// TIA Portal V17 export
// export: Created 2024-08-20T13:26:08.3005341Z, ExportSetting WithDefaults, DisplayName Totally Integrated Automation Portal, DisplayVersion V17 Update 4, DisplayName TIA Portal Openness, DisplayVersion V17 Update 4, DisplayName TIA Portal Version Control Interface, DisplayVersion V17, DisplayName STEP 7 Professional, DisplayVersion V17 Update 4, DisplayName STEP 7 Safety, DisplayVersion V17, DisplayName WinCC Advanced, DisplayVersion V17 Update 4
FUNCTION_BLOCK "INTPRO"   // FB202, LAD
{ S7_Optimized_Access := 'FALSE' }
VERSION : 0.1
// stored: AutoNumber true, IsIECCheckEnabled false, SetENOAutomatically false, UDAEnableTagReadback false
   VAR DB_SPECIFIC
      EE_P_NIV : Bool;   // HAILITA BOMBA PRINCIPAL PELO NÍVEL
      EE_C1_NIV : Bool;   // HAILITA BOMBA COMPLEMENTAR 1 PELO NÍVEL
      EE_C2_NIV : Bool;   // HAILITA BOMBA COMPLEMENTAR 2 PELO NÍVEL
      EE_P_LS : Bool;   // HAILITA BOMBA PRINCIPAL PELAS BÓIAS
      EE_C1_LS : Bool;   // HAILITA BOMBA COMLEMENTAR 1 PELAS BÓIAS
      EE_C2_LS : Bool;   // HAILITA BOMBA COMPLEMENTAR 2 PELAS BÓIAS
      HAB_P_EE : Bool;   // LIGA BOMBA PRINCIPAL DA ELEVATÓRIA
      HAB_C1_EE : Bool;   // LIGA BOMBA COMPLEMENTAR 1 DA ELEVATÓRIA
      HAB_C2_EE : Bool;   // LIGA BOMBA COMPLEMENTAR 2 DA ELEVATÓRIA
      AUXP01 : Bool;
      BS01OK : Bool;
      BS02OK : Bool;
      BS03OK : Bool;
      L_BS01 : Bool;
      L_BS02 : Bool;
      L_BS03 : Bool;
      AUXP02 : Bool;
      AUXP03 : Bool;
      AUXP04 : Bool;
      AUXP05 : Bool;
      AUXP06 : Bool;
      AUXP07 : Bool;
      ETBS01_T001 : Int;
      ETBS02_T001 : Int;
      ETBS03_T001 : Int;
      BS01TO : Int;
      BS02TO : Int;
      BS03TO : Int;
      BS01TEOK : DInt;
      BS02TEOK : DInt;
      BS03TEOK : DInt;
      TE00 { S7_SetPoint := 'True'} : IEC_TIMER;
   END_VAR
   VAR
      RODEE { S7_SetPoint := 'True'} : "ROD4";
   END_VAR
   VAR_TEMP
      T011S : Int;
      ET_TE00 : Time;
   END_VAR
BEGIN

REGION Network 1: Alarme falha de sinal transmissor de nivel
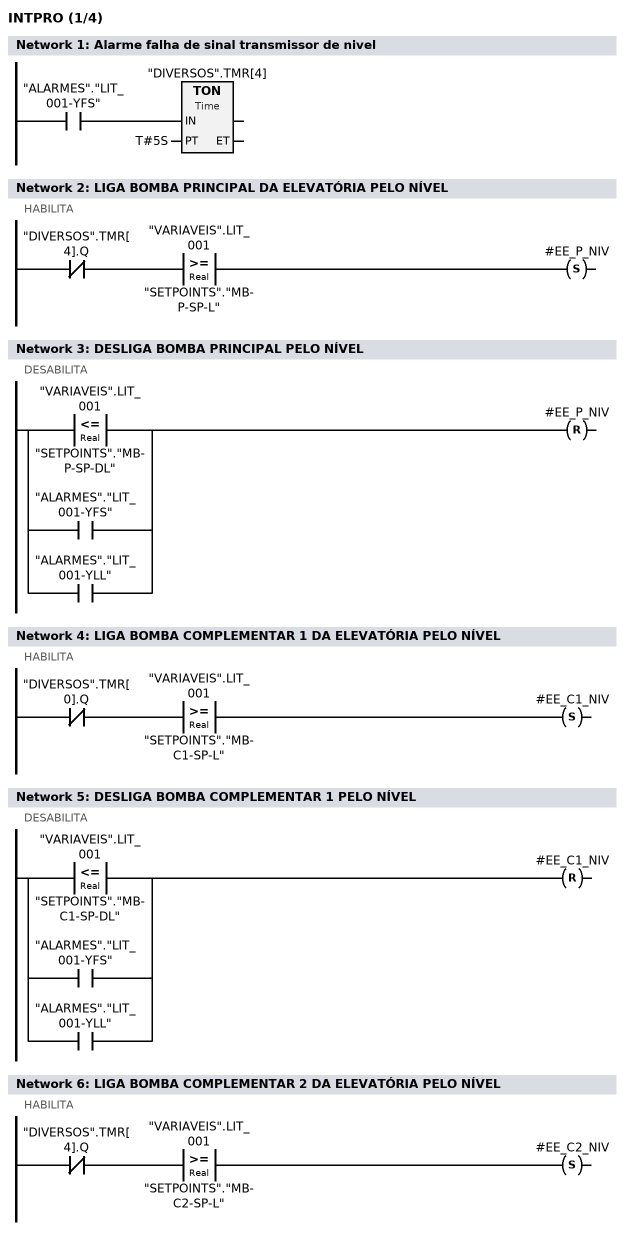
   RUNG wire#powerrail
      Contact( "ALARMES"."LIT_001-YFS" )
      { S7_Templates := "time_type := Time" } "DIVERSOS".TMR[4].TON(pt := T#5S, et =>)
   END_RUNG
   // the same network as SCL:
   "DIVERSOS".TMR[4].TON(IN := "ALARMES"."LIT_001-YFS", PT := T#5S);
END_REGION

REGION Network 2: LIGA BOMBA PRINCIPAL DA ELEVATÓRIA PELO NÍVEL
   // HABILITA
   RUNG wire#powerrail
      I_Contact( "DIVERSOS".TMR[4].Q )
      { S7_Templates := "SrcType := Real" } GE_Contact(in1 := "VARIAVEIS".LIT_001, in2 := "SETPOINTS"."MB-P-SP-L")
      S_Coil( #EE_P_NIV )
   END_RUNG
   // the same network as SCL:
   IF NOT "DIVERSOS".TMR[4].Q AND ("VARIAVEIS".LIT_001 >= "SETPOINTS"."MB-P-SP-L") THEN
       #EE_P_NIV := TRUE;
   END_IF;
END_REGION

REGION Network 3: DESLIGA BOMBA PRINCIPAL PELO NÍVEL
   // DESABILITA
   RUNG wire#powerrail
      { S7_Templates := "SrcType := Real" } LE_Contact(in1 := "VARIAVEIS".LIT_001, in2 := "SETPOINTS"."MB-P-SP-DL")
      wire#w1
      R_Coil( #EE_P_NIV )
   END_RUNG
   RUNG wire#powerrail
      Contact( "ALARMES"."LIT_001-YFS" )
   END_RUNG wire#w1
   RUNG wire#powerrail
      Contact( "ALARMES"."LIT_001-YLL" )
   END_RUNG wire#w1
   // the same network as SCL:
   IF ("VARIAVEIS".LIT_001 <= "SETPOINTS"."MB-P-SP-DL") OR "ALARMES"."LIT_001-YFS" OR "ALARMES"."LIT_001-YLL" THEN
       #EE_P_NIV := FALSE;
   END_IF;
END_REGION

REGION Network 4: LIGA BOMBA COMPLEMENTAR 1 DA ELEVATÓRIA PELO NÍVEL
   // HABILITA
   RUNG wire#powerrail
      I_Contact( "DIVERSOS".TMR[0].Q )
      { S7_Templates := "SrcType := Real" } GE_Contact(in1 := "VARIAVEIS".LIT_001, in2 := "SETPOINTS"."MB-C1-SP-L")
      S_Coil( #EE_C1_NIV )
   END_RUNG
   // the same network as SCL:
   IF NOT "DIVERSOS".TMR[0].Q AND ("VARIAVEIS".LIT_001 >= "SETPOINTS"."MB-C1-SP-L") THEN
       #EE_C1_NIV := TRUE;
   END_IF;
END_REGION

REGION Network 5: DESLIGA BOMBA COMPLEMENTAR 1 PELO NÍVEL
   // DESABILITA
   RUNG wire#powerrail
      { S7_Templates := "SrcType := Real" } LE_Contact(in1 := "VARIAVEIS".LIT_001, in2 := "SETPOINTS"."MB-C1-SP-DL")
      wire#w1
      R_Coil( #EE_C1_NIV )
   END_RUNG
   RUNG wire#powerrail
      Contact( "ALARMES"."LIT_001-YFS" )
   END_RUNG wire#w1
   RUNG wire#powerrail
      Contact( "ALARMES"."LIT_001-YLL" )
   END_RUNG wire#w1
   // the same network as SCL:
   IF ("VARIAVEIS".LIT_001 <= "SETPOINTS"."MB-C1-SP-DL") OR "ALARMES"."LIT_001-YFS" OR "ALARMES"."LIT_001-YLL" THEN
       #EE_C1_NIV := FALSE;
   END_IF;
END_REGION

REGION Network 6: LIGA BOMBA COMPLEMENTAR 2 DA ELEVATÓRIA PELO NÍVEL
   // HABILITA
   RUNG wire#powerrail
      I_Contact( "DIVERSOS".TMR[4].Q )
      { S7_Templates := "SrcType := Real" } GE_Contact(in1 := "VARIAVEIS".LIT_001, in2 := "SETPOINTS"."MB-C2-SP-L")
      S_Coil( #EE_C2_NIV )
   END_RUNG
   // the same network as SCL:
   IF NOT "DIVERSOS".TMR[4].Q AND ("VARIAVEIS".LIT_001 >= "SETPOINTS"."MB-C2-SP-L") THEN
       #EE_C2_NIV := TRUE;
   END_IF;
END_REGION

REGION Network 7: DESLIGA BOMBA COMPLEMENTAR 2 PELO NÍVEL
   // DESABILITA
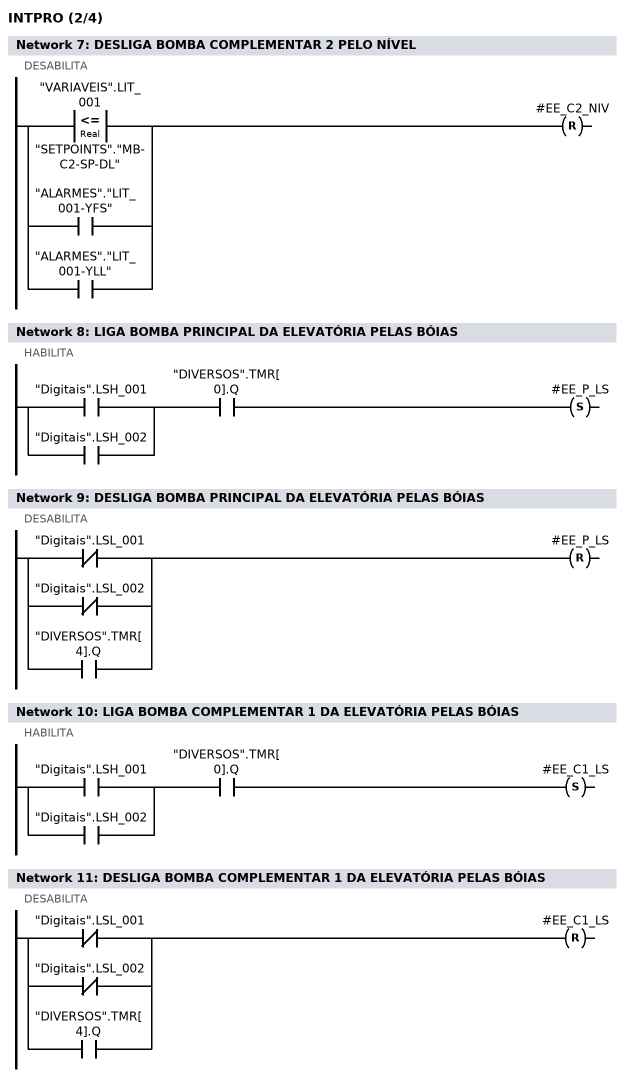
   RUNG wire#powerrail
      { S7_Templates := "SrcType := Real" } LE_Contact(in1 := "VARIAVEIS".LIT_001, in2 := "SETPOINTS"."MB-C2-SP-DL")
      wire#w1
      R_Coil( #EE_C2_NIV )
   END_RUNG
   RUNG wire#powerrail
      Contact( "ALARMES"."LIT_001-YFS" )
   END_RUNG wire#w1
   RUNG wire#powerrail
      Contact( "ALARMES"."LIT_001-YLL" )
   END_RUNG wire#w1
   // the same network as SCL:
   IF ("VARIAVEIS".LIT_001 <= "SETPOINTS"."MB-C2-SP-DL") OR "ALARMES"."LIT_001-YFS" OR "ALARMES"."LIT_001-YLL" THEN
       #EE_C2_NIV := FALSE;
   END_IF;
END_REGION

REGION Network 8: LIGA BOMBA PRINCIPAL DA ELEVATÓRIA PELAS BÓIAS
   // HABILITA
   RUNG wire#powerrail
      Contact( "Digitais".LSH_001 )
      wire#w1
      Contact( "DIVERSOS".TMR[0].Q )
      S_Coil( #EE_P_LS )
   END_RUNG
   RUNG wire#powerrail
      Contact( "Digitais".LSH_002 )
   END_RUNG wire#w1
   // the same network as SCL:
   IF ("Digitais".LSH_001 OR "Digitais".LSH_002) AND "DIVERSOS".TMR[0].Q THEN #EE_P_LS := TRUE; END_IF;
END_REGION

REGION Network 9: DESLIGA BOMBA PRINCIPAL DA ELEVATÓRIA PELAS BÓIAS
   // DESABILITA
   RUNG wire#powerrail
      I_Contact( "Digitais".LSL_001 )
      wire#w1
      R_Coil( #EE_P_LS )
   END_RUNG
   RUNG wire#powerrail
      I_Contact( "Digitais".LSL_002 )
   END_RUNG wire#w1
   RUNG wire#powerrail
      Contact( "DIVERSOS".TMR[4].Q )
   END_RUNG wire#w1
   // the same network as SCL:
   IF NOT "Digitais".LSL_001 OR NOT "Digitais".LSL_002 OR "DIVERSOS".TMR[4].Q THEN #EE_P_LS := FALSE; END_IF;
END_REGION

REGION Network 10: LIGA BOMBA COMPLEMENTAR 1 DA ELEVATÓRIA PELAS BÓIAS
   // HABILITA
   RUNG wire#powerrail
      Contact( "Digitais".LSH_001 )
      wire#w1
      Contact( "DIVERSOS".TMR[0].Q )
      S_Coil( #EE_C1_LS )
   END_RUNG
   RUNG wire#powerrail
      Contact( "Digitais".LSH_002 )
   END_RUNG wire#w1
   // the same network as SCL:
   IF ("Digitais".LSH_001 OR "Digitais".LSH_002) AND "DIVERSOS".TMR[0].Q THEN #EE_C1_LS := TRUE; END_IF;
END_REGION

REGION Network 11: DESLIGA BOMBA COMPLEMENTAR 1 DA ELEVATÓRIA PELAS BÓIAS
   // DESABILITA
   RUNG wire#powerrail
      I_Contact( "Digitais".LSL_001 )
      wire#w1
      R_Coil( #EE_C1_LS )
   END_RUNG
   RUNG wire#powerrail
      I_Contact( "Digitais".LSL_002 )
   END_RUNG wire#w1
   RUNG wire#powerrail
      Contact( "DIVERSOS".TMR[4].Q )
   END_RUNG wire#w1
   // the same network as SCL:
   IF NOT "Digitais".LSL_001 OR NOT "Digitais".LSL_002 OR "DIVERSOS".TMR[4].Q THEN
       #EE_C1_LS := FALSE;
   END_IF;
END_REGION

REGION Network 12: LIGA BOMBA COMPLEMENTAR 2 DA ELEVATÓRIA PELAS BÓIAS
   // HABILITA
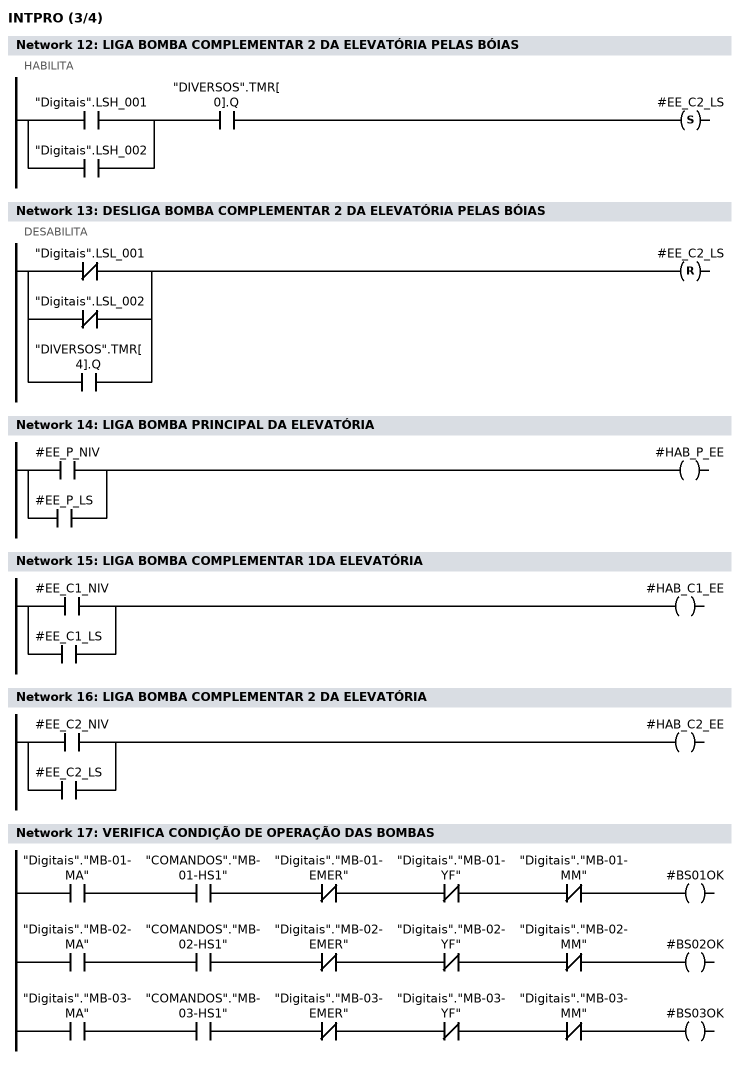
   RUNG wire#powerrail
      Contact( "Digitais".LSH_001 )
      wire#w1
      Contact( "DIVERSOS".TMR[0].Q )
      S_Coil( #EE_C2_LS )
   END_RUNG
   RUNG wire#powerrail
      Contact( "Digitais".LSH_002 )
   END_RUNG wire#w1
   // the same network as SCL:
   IF ("Digitais".LSH_001 OR "Digitais".LSH_002) AND "DIVERSOS".TMR[0].Q THEN #EE_C2_LS := TRUE; END_IF;
END_REGION

REGION Network 13: DESLIGA BOMBA COMPLEMENTAR 2 DA ELEVATÓRIA PELAS BÓIAS
   // DESABILITA
   RUNG wire#powerrail
      I_Contact( "Digitais".LSL_001 )
      wire#w1
      R_Coil( #EE_C2_LS )
   END_RUNG
   RUNG wire#powerrail
      I_Contact( "Digitais".LSL_002 )
   END_RUNG wire#w1
   RUNG wire#powerrail
      Contact( "DIVERSOS".TMR[4].Q )
   END_RUNG wire#w1
   // the same network as SCL:
   IF NOT "Digitais".LSL_001 OR NOT "Digitais".LSL_002 OR "DIVERSOS".TMR[4].Q THEN
       #EE_C2_LS := FALSE;
   END_IF;
END_REGION

REGION Network 14: LIGA BOMBA PRINCIPAL DA ELEVATÓRIA
   RUNG wire#powerrail
      Contact( #EE_P_NIV )
      wire#w1
      Coil( #HAB_P_EE )
   END_RUNG
   RUNG wire#powerrail
      Contact( #EE_P_LS )
   END_RUNG wire#w1
   // the same network as SCL:
   #HAB_P_EE := #EE_P_NIV OR #EE_P_LS;
END_REGION

REGION Network 15: LIGA BOMBA COMPLEMENTAR 1DA ELEVATÓRIA
   RUNG wire#powerrail
      Contact( #EE_C1_NIV )
      wire#w1
      Coil( #HAB_C1_EE )
   END_RUNG
   RUNG wire#powerrail
      Contact( #EE_C1_LS )
   END_RUNG wire#w1
   // the same network as SCL:
   #HAB_C1_EE := #EE_C1_NIV OR #EE_C1_LS;
END_REGION

REGION Network 16: LIGA BOMBA COMPLEMENTAR 2 DA ELEVATÓRIA
   RUNG wire#powerrail
      Contact( #EE_C2_NIV )
      wire#w1
      Coil( #HAB_C2_EE )
   END_RUNG
   RUNG wire#powerrail
      Contact( #EE_C2_LS )
   END_RUNG wire#w1
   // the same network as SCL:
   #HAB_C2_EE := #EE_C2_NIV OR #EE_C2_LS;
END_REGION

REGION Network 17: VERIFICA CONDIÇÃO DE OPERAÇÃO DAS BOMBAS
   RUNG wire#powerrail
      Contact( "Digitais"."MB-01-MA" )
      Contact( "COMANDOS"."MB-01-HS1" )
      I_Contact( "Digitais"."MB-01-EMER" )
      I_Contact( "Digitais"."MB-01-YF" )
      I_Contact( "Digitais"."MB-01-MM" )
      Coil( #BS01OK )
   END_RUNG
   RUNG wire#powerrail
      Contact( "Digitais"."MB-02-MA" )
      Contact( "COMANDOS"."MB-02-HS1" )
      I_Contact( "Digitais"."MB-02-EMER" )
      I_Contact( "Digitais"."MB-02-YF" )
      I_Contact( "Digitais"."MB-02-MM" )
      Coil( #BS02OK )
   END_RUNG
   RUNG wire#powerrail
      Contact( "Digitais"."MB-03-MA" )
      Contact( "COMANDOS"."MB-03-HS1" )
      I_Contact( "Digitais"."MB-03-EMER" )
      I_Contact( "Digitais"."MB-03-YF" )
      I_Contact( "Digitais"."MB-03-MM" )
      Coil( #BS03OK )
   END_RUNG
   // the same network as SCL:
   #BS01OK := "Digitais"."MB-01-MA" AND "COMANDOS"."MB-01-HS1" AND NOT "Digitais"."MB-01-EMER" AND NOT "Digitais"."MB-01-YF" AND NOT "Digitais"."MB-01-MM";
   #BS02OK := "Digitais"."MB-02-MA" AND "COMANDOS"."MB-02-HS1" AND NOT "Digitais"."MB-02-EMER" AND NOT "Digitais"."MB-02-YF" AND NOT "Digitais"."MB-02-MM";
   #BS03OK := "Digitais"."MB-03-MA" AND "COMANDOS"."MB-03-HS1" AND NOT "Digitais"."MB-03-EMER" AND NOT "Digitais"."MB-03-YF" AND NOT "Digitais"."MB-03-MM";
END_REGION

REGION Network 18: RODÍZIO DAS BOMBAS
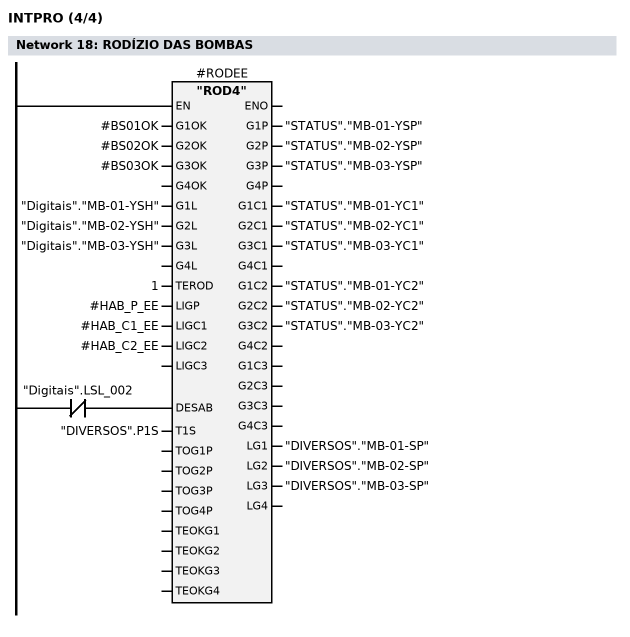
   RUNG wire#powerrail
      #RODEE(DESAB := wire#w1, G1OK := #BS01OK, G2OK := #BS02OK, G3OK := #BS03OK, G4OK :=, G1L := "Digitais"."MB-01-YSH", G2L := "Digitais"."MB-02-YSH", G3L := "Digitais"."MB-03-YSH", G4L :=, TEROD := 1, LIGP := #HAB_P_EE, LIGC1 := #HAB_C1_EE, LIGC2 := #HAB_C2_EE, LIGC3 :=, T1S := "DIVERSOS".P1S, TOG1P :=, TOG2P :=, TOG3P :=, TOG4P :=, TEOKG1 :=, TEOKG2 :=, TEOKG3 :=, TEOKG4 :=, G1P => "STATUS"."MB-01-YSP", G2P => "STATUS"."MB-02-YSP", G3P => "STATUS"."MB-03-YSP", G4P =>, G1C1 => "STATUS"."MB-01-YC1", G2C1 => "STATUS"."MB-02-YC1", G3C1 => "STATUS"."MB-03-YC1", G4C1 =>, G1C2 => "STATUS"."MB-01-YC2", G2C2 => "STATUS"."MB-02-YC2", G3C2 => "STATUS"."MB-03-YC2", G4C2 =>, G1C3 =>, G2C3 =>, G3C3 =>, G4C3 =>, LG1 => "DIVERSOS"."MB-01-SP", LG2 => "DIVERSOS"."MB-02-SP", LG3 => "DIVERSOS"."MB-03-SP", LG4 =>)
   END_RUNG
   RUNG wire#powerrail
      I_Contact( "Digitais".LSL_002 )
   END_RUNG wire#w1
   // the same network as SCL:
   #RODEE(G1OK := #BS01OK,   // "ROD4"
          G2OK := #BS02OK,
          G3OK := #BS03OK,
          G1L := "Digitais"."MB-01-YSH",
          G2L := "Digitais"."MB-02-YSH",
          G3L := "Digitais"."MB-03-YSH",
          TEROD := 1,
          LIGP := #HAB_P_EE,
          LIGC1 := #HAB_C1_EE,
          LIGC2 := #HAB_C2_EE,
          DESAB := NOT "Digitais".LSL_002,
          T1S := "DIVERSOS".P1S,
          G1P => "STATUS"."MB-01-YSP",
          G2P => "STATUS"."MB-02-YSP",
          G3P => "STATUS"."MB-03-YSP",
          G1C1 => "STATUS"."MB-01-YC1",
          G2C1 => "STATUS"."MB-02-YC1",
          G3C1 => "STATUS"."MB-03-YC1",
          G1C2 => "STATUS"."MB-01-YC2",
          G2C2 => "STATUS"."MB-02-YC2",
          G3C2 => "STATUS"."MB-03-YC2",
          LG1 => "DIVERSOS"."MB-01-SP",
          LG2 => "DIVERSOS"."MB-02-SP",
          LG3 => "DIVERSOS"."MB-03-SP");
END_REGION
END_FUNCTION_BLOCK
